{attribute 'linkalways'} 
{attribute 'no_explicit_call' := 'This FB is a CLASS and must be accessed using methods or properties'}
{attribute 'enable_dynamic_creation'}
FUNCTION_BLOCK Parameter EXTENDS Disposable IMPLEMENTS I_Parameter
VAR
	_name : T_MAXSTRING;
	_data : I_Datatype;
	_parent : I_HostParameters;
END_VAR

METHOD PUBLIC Accept
VAR_INPUT
	Visitor : I_ParameterVisitor;
END_VAR
Visitor.VisitParameter(this^);
END_METHOD

PROPERTY PUBLIC Data : I_Datatype
GET
Data := _data;
END_GET
END_PROPERTY

METHOD FB_init : BOOL
VAR_INPUT
	bInitRetains : BOOL; // if TRUE, the retain variables are initialized (warm start / cold start)
	bInCopyCode : BOOL;  // if TRUE, the instance afterwards gets moved into the copy code (online change)
	Name : T_MAXSTRING;
	Data : I_Datatype;
	Parent : I_HostParameters;
END_VAR
_name := Name;
_data := Data;
RegisterWithParent(Parent);
END_METHOD

PROPERTY PUBLIC Name : T_MAXSTRING
GET
Name := _name;
END_GET
END_PROPERTY

PROPERTY PUBLIC Parent : I_HostParameters
GET
Parent := _parent;
END_GET
END_PROPERTY

METHOD PUBLIC RegisterWithParent
VAR_INPUT
	Parent : I_HostParameters;
END_VAR
IF Parent = 0 THEN
	RETURN;
END_IF

THIS^._parent := Parent;
Parent.AddParameter(THIS^);
END_METHOD

METHOD PUBLIC SerializeWith
VAR_INPUT
	Serializer : I_Serializer;
END_VAR
Serializer.StartObject();
Serializer.AddKeyString('name',_name);
Serializer.Addkey('datatype');
_data.SerializeTypeWith(Serializer);
Serializer.AddkeyObject('value',_data);
Serializer.EndObject();
END_METHOD

METHOD PUBLIC TryDeserializeFrom : BOOL
VAR_INPUT
	Deserializer : I_Deserializer;
END_VAR
// check name = prameter name


TryDeserializeFrom := _data.TryDeserializeFrom(Deserializer);
END_METHOD

END_FUNCTION_BLOCK

(* stored: Version 1.1.0.1, ProductVersion 3.1.4024.12
   POU Parameter: Id {eaa0ca54-0a21-0aaf-1dd9-4878564e4f5c}, SpecialFunc None
   Folder Constructor: Id {487ef031-4058-0af2-31e5-5368e5c22e10}
   Method Accept: Id {e53d7527-03af-0f69-17de-4a094df11b20}
   Property Data: Id {65957ab6-6ee1-024b-1dde-997589c13367}
   Get Get: Id {8cff9333-d85d-0ca7-1ef2-0b421589b885}
   Method FB_init: Id {3643b8c3-bcdc-0605-199f-bf59b2780fc1}
   Property Name: Id {4a6318e3-2929-0259-19a0-92be35ce16d0}
   Get Get: Id {395bcf64-d6f3-0913-1694-5b849228d9a0}
   Property Parent: Id {6b0a082d-80dd-00ef-195c-b9646bd55928}
   Get Get: Id {3499ec4d-2af4-0aeb-2b55-87ff5f69f0a4}
   Method RegisterWithParent: Id {e6a0eede-b688-0c24-2f67-e84feed89ceb}
   Method SerializeWith: Id {5e3ea962-87a5-4ecc-9bc5-4626e13acdcc}
   Method TryDeserializeFrom: Id {0d32f2cc-8731-4442-b7e6-8584eb88345b} *)
